PROGRAM MAIN
VAR
END_VAR

END_PROGRAM

(* stored: Version 1.1.0.1
   POU MAIN: Id {020d1cff-9f22-4cff-8b05-a70d8068ca5d} *)
